PROGRAM Stn055_20_StorageBreakStopsGrn
VAR
	
	//Note that breakstop 1 is controlled by 3 lane swtich so although called a break stop it is not mapped here
	// Remove these outputs temp to avoid common valve bank conflict for control of outputs with station 51
	//	.fbBreakStop[42].oStopLower :=  <0,1,0>TIIB[N13S00 (AL1332)]^N13S02 (EX260)^RxPDO^output byte 0;
	//	.fbBreakStop[43].oStopLower :=  <0,1,1>TIIB[N13S00 (AL1332)]^N13S02 (EX260)^RxPDO^output byte 0'
	
	{attribute 'TcLinkToOSO' := '.fbBreakStop[2].iBufferFull :=  <0,1,1>TIIB[N62S00 (AL1332)]^N62S03 (AL2341)^TxPDO^input byte 2;
		.fbBreakStop[2].iPuckPresent :=  <0,1,1>TIIB[N62S00 (AL1332)]^N62S03 (AL2341)^TxPDO^input byte 0;
		.fbBreakStop[2].oStopLower :=  <0,1,4>TIIB[N62S00 (AL1332)]^N62S02 (EX260)^RxPDO^output byte 0;
		.fbBreakStop[3].iBufferFull :=  <0,1,0>TIIB[N62S00 (AL1332)]^N62S05 (AL2341)^TxPDO^input byte 2;
		.fbBreakStop[3].iPuckPresent :=  <0,1,0>TIIB[N62S00 (AL1332)]^N62S05 (AL2341)^TxPDO^input byte 0;
		.fbBreakStop[3].oStopLower :=  <0,1,5>TIIB[N62S00 (AL1332)]^N62S02 (EX260)^RxPDO^output byte 0;
		.fbBreakStop[4].iBufferFull :=  <0,1,0>TIIB[N66S00 (AL1332)]^N66S01 (AL2341)^TxPDO^input byte 2;
		.fbBreakStop[4].iPuckPresent :=  <0,1,0>TIIB[N66S00 (AL1332)]^N66S01 (AL2341)^TxPDO^input byte 0;
		.fbBreakStop[4].oStopLower :=  <0,1,0>TIIB[N66S00 (AL1332)]^N66S02 (EX260)^RxPDO^output byte 0;
		.fbBreakStop[5].iBufferFull :=  <0,1,1>TIIB[N66S00 (AL1332)]^N66S01 (AL2341)^TxPDO^input byte 2;
		.fbBreakStop[5].iPuckPresent :=  <0,1,1>TIIB[N66S00 (AL1332)]^N66S01 (AL2341)^TxPDO^input byte 0;
		.fbBreakStop[5].oStopLower :=  <0,1,1>TIIB[N66S00 (AL1332)]^N66S02 (EX260)^RxPDO^output byte 0;
		.fbBreakStop[6].iBufferFull :=  <0,1,2>TIIB[N66S00 (AL1332)]^N66S01 (AL2341)^TxPDO^input byte 2;
		.fbBreakStop[6].iPuckPresent :=  <0,1,2>TIIB[N66S00 (AL1332)]^N66S01 (AL2341)^TxPDO^input byte 0;
		.fbBreakStop[6].oStopLower :=  <0,1,2>TIIB[N66S00 (AL1332)]^N66S02 (EX260)^RxPDO^output byte 0;
		.fbBreakStop[7].iBufferFull :=  <0,1,0>TIIB[N66S00 (AL1332)]^N66S03 (AL2341)^TxPDO^input byte 2;
		.fbBreakStop[7].iPuckPresent :=  <0,1,0>TIIB[N66S00 (AL1332)]^N66S03 (AL2341)^TxPDO^input byte 0;
		.fbBreakStop[7].oStopLower :=  <0,1,3>TIIB[N66S00 (AL1332)]^N66S02 (EX260)^RxPDO^output byte 0;
		.fbBreakStop[8].iBufferFull :=  <0,1,1>TIIB[N66S00 (AL1332)]^N66S03 (AL2341)^TxPDO^input byte 2;
		.fbBreakStop[8].iPuckPresent :=  <0,1,1>TIIB[N66S00 (AL1332)]^N66S03 (AL2341)^TxPDO^input byte 0;
		.fbBreakStop[8].oStopLower :=  <0,1,4>TIIB[N66S00 (AL1332)]^N66S02 (EX260)^RxPDO^output byte 0;
		.fbBreakStop[9].iBufferFull :=  <0,1,2>TIIB[N66S00 (AL1332)]^N66S03 (AL2341)^TxPDO^input byte 2;
		.fbBreakStop[9].iPuckPresent :=  <0,1,2>TIIB[N66S00 (AL1332)]^N66S03 (AL2341)^TxPDO^input byte 0;
		.fbBreakStop[9].oStopLower :=  <0,1,5>TIIB[N66S00 (AL1332)]^N66S02 (EX260)^RxPDO^output byte 0;
		.fbBreakStop[10].iBufferFull :=  <0,1,3>TIIB[N66S00 (AL1332)]^N66S03 (AL2341)^TxPDO^input byte 2;
		.fbBreakStop[10].iPuckPresent :=  <0,1,3>TIIB[N66S00 (AL1332)]^N66S03 (AL2341)^TxPDO^input byte 0;
		.fbBreakStop[10].oStopLower :=  <0,1,6>TIIB[N66S00 (AL1332)]^N66S02 (EX260)^RxPDO^output byte 0;
		.fbBreakStop[11].iBufferFull :=  <0,1,0>TIIB[N67S00 (AL1332)]^N67S01 (AL2341)^TxPDO^input byte 2;
		.fbBreakStop[11].iPuckPresent :=  <0,1,0>TIIB[N67S00 (AL1332)]^N67S01 (AL2341)^TxPDO^input byte 0;
		.fbBreakStop[11].oStopLower :=  <0,1,0>TIIB[N67S00 (AL1332)]^N67S02 (EX260)^RxPDO^output byte 0;
		.fbBreakStop[12].iBufferFull :=  <0,1,1>TIIB[N67S00 (AL1332)]^N67S01 (AL2341)^TxPDO^input byte 2;
		.fbBreakStop[12].iPuckPresent :=  <0,1,1>TIIB[N67S00 (AL1332)]^N67S01 (AL2341)^TxPDO^input byte 0;
		.fbBreakStop[12].oStopLower :=  <0,1,1>TIIB[N67S00 (AL1332)]^N67S02 (EX260)^RxPDO^output byte 0;
		.fbBreakStop[13].iBufferFull :=  <0,1,0>TIIB[N67S00 (AL1332)]^N67S01 (AL2341)^TxPDO^input byte 3;
		.fbBreakStop[13].iPuckPresent :=  <0,1,0>TIIB[N67S00 (AL1332)]^N67S01 (AL2341)^TxPDO^input byte 1;
		.fbBreakStop[13].oStopLower :=  <0,1,3>TIIB[N67S00 (AL1332)]^N67S02 (EX260)^RxPDO^output byte 0;
		.fbBreakStop[14].iBufferFull :=  <0,1,1>TIIB[N67S00 (AL1332)]^N67S01 (AL2341)^TxPDO^input byte 3;
		.fbBreakStop[14].iPuckPresent :=  <0,1,1>TIIB[N67S00 (AL1332)]^N67S01 (AL2341)^TxPDO^input byte 1;
		.fbBreakStop[14].oStopLower :=  <0,1,6>TIIB[N67S00 (AL1332)]^N67S02 (EX260)^RxPDO^output byte 0;
		.fbBreakStop[15].iBufferFull :=  <0,1,2>TIIB[N67S00 (AL1332)]^N67S01 (AL2341)^TxPDO^input byte 3;
		.fbBreakStop[15].iPuckPresent :=  <0,1,2>TIIB[N67S00 (AL1332)]^N67S01 (AL2341)^TxPDO^input byte 1;
		.fbBreakStop[15].oStopLower :=  <0,1,7>TIIB[N67S00 (AL1332)]^N67S02 (EX260)^RxPDO^output byte 0;
		.fbBreakStop[16].iBufferFull :=  <0,1,4>TIIB[N67S00 (AL1332)]^N67S03 (AL2341)^TxPDO^input byte 2;
		.fbBreakStop[16].iPuckPresent :=  <0,1,4>TIIB[N67S00 (AL1332)]^N67S03 (AL2341)^TxPDO^input byte 0;
		.fbBreakStop[16].oStopLower :=  <0,1,4>TIIB[N67S00 (AL1332)]^N67S02 (EX260)^RxPDO^output byte 1;
		.fbBreakStop[17].iBufferFull :=  <0,1,1>TIIB[N67S00 (AL1332)]^N67S03 (AL2341)^TxPDO^input byte 3;
		.fbBreakStop[17].iPuckPresent :=  <0,1,1>TIIB[N67S00 (AL1332)]^N67S03 (AL2341)^TxPDO^input byte 1;
		.fbBreakStop[17].oStopLower :=  <0,1,5>TIIB[N67S00 (AL1332)]^N67S02 (EX260)^RxPDO^output byte 1;
		.fbBreakStop[18].iBufferFull :=  <0,1,2>TIIB[N67S00 (AL1332)]^N67S03 (AL2341)^TxPDO^input byte 3;
		.fbBreakStop[18].iPuckPresent :=  <0,1,2>TIIB[N67S00 (AL1332)]^N67S03 (AL2341)^TxPDO^input byte 1;
		.fbBreakStop[18].oStopLower :=  <0,1,0>TIIB[N67S00 (AL1332)]^N67S02 (EX260)^RxPDO^output byte 2;
		.fbBreakStop[19].iBufferFull :=  <0,1,0>TIIB[N67S00 (AL1332)]^N67S05 (AL2341)^TxPDO^input byte 2;
		.fbBreakStop[19].iPuckPresent :=  <0,1,0>TIIB[N67S00 (AL1332)]^N67S05 (AL2341)^TxPDO^input byte 0;
		.fbBreakStop[19].oStopLower :=  <0,1,1>TIIB[N67S00 (AL1332)]^N67S02 (EX260)^RxPDO^output byte 2;
		.fbBreakStop[20].iBufferFull :=  <0,1,1>TIIB[N67S00 (AL1332)]^N67S05 (AL2341)^TxPDO^input byte 2;
		.fbBreakStop[20].iPuckPresent :=  <0,1,1>TIIB[N67S00 (AL1332)]^N67S05 (AL2341)^TxPDO^input byte 0;
		.fbBreakStop[20].oStopLower :=  <0,1,2>TIIB[N67S00 (AL1332)]^N67S02 (EX260)^RxPDO^output byte 2;
		.fbBreakStop[21].iBufferFull :=  <0,1,2>TIIB[N67S00 (AL1332)]^N67S05 (AL2341)^TxPDO^input byte 2;
		.fbBreakStop[21].iPuckPresent :=  <0,1,2>TIIB[N67S00 (AL1332)]^N67S05 (AL2341)^TxPDO^input byte 0;
		.fbBreakStop[21].oStopLower :=  <0,1,3>TIIB[N67S00 (AL1332)]^N67S02 (EX260)^RxPDO^output byte 2;
		.fbBreakStop[22].iBufferFull :=  <0,1,4>TIIB[N67S00 (AL1332)]^N67S05 (AL2341)^TxPDO^input byte 2;
		.fbBreakStop[22].iPuckPresent :=  <0,1,4>TIIB[N67S00 (AL1332)]^N67S05 (AL2341)^TxPDO^input byte 0;
		.fbBreakStop[22].oStopLower :=  <0,1,6>TIIB[N67S00 (AL1332)]^N67S02 (EX260)^RxPDO^output byte 2;
		.fbBreakStop[23].iBufferFull :=  <0,1,0>TIIB[N67S00 (AL1332)]^N67S05 (AL2341)^TxPDO^input byte 3;
		.fbBreakStop[23].iPuckPresent :=  <0,1,0>TIIB[N67S00 (AL1332)]^N67S05 (AL2341)^TxPDO^input byte 1;
		.fbBreakStop[23].oStopLower :=  <0,1,7>TIIB[N67S00 (AL1332)]^N67S02 (EX260)^RxPDO^output byte 2;
		.fbBreakStop[24].iBufferFull :=  <0,1,0>TIIB[N66S00 (AL1332)]^N66S05 (AL2341)^TxPDO^input byte 2;
		.fbBreakStop[24].iPuckPresent :=  <0,1,0>TIIB[N66S00 (AL1332)]^N66S05 (AL2341)^TxPDO^input byte 0;
		.fbBreakStop[24].oStopLower :=  <0,1,0>TIIB[N66S00 (AL1332)]^N66S04 (EX260)^RxPDO^output byte 0;
		.fbBreakStop[25].iBufferFull :=  <0,1,1>TIIB[N66S00 (AL1332)]^N66S05 (AL2341)^TxPDO^input byte 2;
		.fbBreakStop[25].iPuckPresent :=  <0,1,1>TIIB[N66S00 (AL1332)]^N66S05 (AL2341)^TxPDO^input byte 0;
		.fbBreakStop[25].oStopLower :=  <0,1,1>TIIB[N66S00 (AL1332)]^N66S04 (EX260)^RxPDO^output byte 0;
		.fbBreakStop[26].iBufferFull :=  <0,1,2>TIIB[N66S00 (AL1332)]^N66S05 (AL2341)^TxPDO^input byte 2;
		.fbBreakStop[26].iPuckPresent :=  <0,1,2>TIIB[N66S00 (AL1332)]^N66S05 (AL2341)^TxPDO^input byte 0;
		.fbBreakStop[26].oStopLower :=  <0,1,2>TIIB[N66S00 (AL1332)]^N66S04 (EX260)^RxPDO^output byte 0;
		.fbBreakStop[27].iBufferFull :=  <0,1,0>TIIB[N66S00 (AL1332)]^N66S07 (AL2341)^TxPDO^input byte 2;
		.fbBreakStop[27].iPuckPresent :=  <0,1,0>TIIB[N66S00 (AL1332)]^N66S07 (AL2341)^TxPDO^input byte 0;
		.fbBreakStop[27].oStopLower :=  <0,1,3>TIIB[N66S00 (AL1332)]^N66S04 (EX260)^RxPDO^output byte 0;
		.fbBreakStop[28].iBufferFull :=  <0,1,1>TIIB[N66S00 (AL1332)]^N66S07 (AL2341)^TxPDO^input byte 2;
		.fbBreakStop[28].iPuckPresent :=  <0,1,1>TIIB[N66S00 (AL1332)]^N66S07 (AL2341)^TxPDO^input byte 0;
		.fbBreakStop[28].oStopLower :=  <0,1,4>TIIB[N66S00 (AL1332)]^N66S04 (EX260)^RxPDO^output byte 0;
		.fbBreakStop[29].iBufferFull :=  <0,1,0>TIIB[N71S00 (AL1332)]^N71S01 (AL2341)^TxPDO^input byte 2;
		.fbBreakStop[29].iPuckPresent :=  <0,1,0>TIIB[N71S00 (AL1332)]^N71S01 (AL2341)^TxPDO^input byte 0;
		.fbBreakStop[29].oStopLower :=  <0,1,0>TIIB[N71S00 (AL1332)]^N71S02 (EX260)^RxPDO^output byte 0;
		.fbBreakStop[30].iBufferFull :=  <0,1,1>TIIB[N71S00 (AL1332)]^N71S01 (AL2341)^TxPDO^input byte 2;
		.fbBreakStop[30].iPuckPresent :=  <0,1,1>TIIB[N71S00 (AL1332)]^N71S01 (AL2341)^TxPDO^input byte 0;
		.fbBreakStop[30].oStopLower :=  <0,1,1>TIIB[N71S00 (AL1332)]^N71S02 (EX260)^RxPDO^output byte 0;
		.fbBreakStop[31].iBufferFull :=  <0,1,0>TIIB[N71S00 (AL1332)]^N71S03 (AL2341)^TxPDO^input byte 2;
		.fbBreakStop[31].iPuckPresent :=  <0,1,0>TIIB[N71S00 (AL1332)]^N71S03 (AL2341)^TxPDO^input byte 0;
		.fbBreakStop[31].oStopLower :=  <0,1,2>TIIB[N71S00 (AL1332)]^N71S02 (EX260)^RxPDO^output byte 0;
		.fbBreakStop[32].iBufferFull :=  <0,1,1>TIIB[N71S00 (AL1332)]^N71S03 (AL2341)^TxPDO^input byte 2;
		.fbBreakStop[32].iPuckPresent :=  <0,1,1>TIIB[N71S00 (AL1332)]^N71S03 (AL2341)^TxPDO^input byte 0;
		.fbBreakStop[32].oStopLower :=  <0,1,3>TIIB[N71S00 (AL1332)]^N71S02 (EX260)^RxPDO^output byte 0;
		.fbBreakStop[33].iBufferFull :=  <0,1,0>TIIB[N71S00 (AL1332)]^N71S05 (AL2341)^TxPDO^input byte 2;
		.fbBreakStop[33].iPuckPresent :=  <0,1,0>TIIB[N71S00 (AL1332)]^N71S05 (AL2341)^TxPDO^input byte 0;
		.fbBreakStop[33].oStopLower :=  <0,1,4>TIIB[N71S00 (AL1332)]^N71S02 (EX260)^RxPDO^output byte 0;
		.fbBreakStop[34].iBufferFull :=  <0,1,1>TIIB[N71S00 (AL1332)]^N71S05 (AL2341)^TxPDO^input byte 2;
		.fbBreakStop[34].iPuckPresent :=  <0,1,1>TIIB[N71S00 (AL1332)]^N71S05 (AL2341)^TxPDO^input byte 0;
		.fbBreakStop[34].oStopLower :=  <0,1,5>TIIB[N71S00 (AL1332)]^N71S02 (EX260)^RxPDO^output byte 0;
		.fbBreakStop[35].iBufferFull :=  <0,1,0>TIIB[N73S00 (AL1332)]^N73S01 (AL2341)^TxPDO^input byte 2;
		.fbBreakStop[35].iPuckPresent :=  <0,1,0>TIIB[N73S00 (AL1332)]^N73S01 (AL2341)^TxPDO^input byte 0;
		.fbBreakStop[35].oStopLower :=  <0,1,0>TIIB[N73S00 (AL1332)]^N73S02 (EX260)^RxPDO^output byte 0;
		.fbBreakStop[36].iBufferFull :=  <0,1,1>TIIB[N73S00 (AL1332)]^N73S01 (AL2341)^TxPDO^input byte 2;
		.fbBreakStop[36].iPuckPresent :=  <0,1,1>TIIB[N73S00 (AL1332)]^N73S01 (AL2341)^TxPDO^input byte 0;
		.fbBreakStop[36].oStopLower :=  <0,1,1>TIIB[N73S00 (AL1332)]^N73S02 (EX260)^RxPDO^output byte 0;
		.fbBreakStop[37].iBufferFull :=  <0,1,0>TIIB[N73S00 (AL1332)]^N73S03 (AL2341)^TxPDO^input byte 2;
		.fbBreakStop[37].iPuckPresent :=  <0,1,0>TIIB[N73S00 (AL1332)]^N73S03 (AL2341)^TxPDO^input byte 0;
		.fbBreakStop[37].oStopLower :=  <0,1,2>TIIB[N73S00 (AL1332)]^N73S02 (EX260)^RxPDO^output byte 0;
		.fbBreakStop[38].iBufferFull :=  <0,1,1>TIIB[N73S00 (AL1332)]^N73S03 (AL2341)^TxPDO^input byte 2;
		.fbBreakStop[38].iPuckPresent :=  <0,1,1>TIIB[N73S00 (AL1332)]^N73S03 (AL2341)^TxPDO^input byte 0;
		.fbBreakStop[38].oStopLower :=  <0,1,3>TIIB[N73S00 (AL1332)]^N73S02 (EX260)^RxPDO^output byte 0;
		.fbBreakStop[39].iBufferFull :=  <0,1,2>TIIB[N73S00 (AL1332)]^N73S03 (AL2341)^TxPDO^input byte 2;
		.fbBreakStop[39].iPuckPresent :=  <0,1,2>TIIB[N73S00 (AL1332)]^N73S03 (AL2341)^TxPDO^input byte 0;
		.fbBreakStop[39].oStopLower :=  <0,1,4>TIIB[N73S00 (AL1332)]^N73S02 (EX260)^RxPDO^output byte 0;
		.fbBreakStop[40].iBufferFull :=  <0,1,0>TIIB[N73S00 (AL1332)]^N73S05 (AL2341)^TxPDO^input byte 2;
		.fbBreakStop[40].iPuckPresent :=  <0,1,0>TIIB[N73S00 (AL1332)]^N73S05 (AL2341)^TxPDO^input byte 0;
		.fbBreakStop[40].oStopLower :=  <0,1,5>TIIB[N73S00 (AL1332)]^N73S02 (EX260)^RxPDO^output byte 0;
		.fbBreakStop[41].iBufferFull :=  <0,1,1>TIIB[N73S00 (AL1332)]^N73S05 (AL2341)^TxPDO^input byte 2;
		.fbBreakStop[41].iPuckPresent :=  <0,1,1>TIIB[N73S00 (AL1332)]^N73S05 (AL2341)^TxPDO^input byte 0;
		.fbBreakStop[41].oStopLower :=  <0,1,6>TIIB[N73S00 (AL1332)]^N73S02 (EX260)^RxPDO^output byte 0;
		.fbBreakStop[42].iBufferFull :=  <0,1,0>TIIB[N12S00 (AL1332)]^N12S07 (AL2341)^TxPDO^input byte 2;
		.fbBreakStop[42].iPuckPresent :=  <0,1,0>TIIB[N12S00 (AL1332)]^N12S07 (AL2341)^TxPDO^input byte 0;
		.fbBreakStop[43].iBufferFull :=  <0,1,0>TIIB[N13S00 (AL1332)]^N13S01 (AL2341)^TxPDO^input byte 2;
		.fbBreakStop[43].iPuckPresent :=  <0,1,0>TIIB[N13S00 (AL1332)]^N13S01 (AL2341)^TxPDO^input byte 0'}
	fbBreakStopGroup: FB_BreakStopGroup;
	
	i: DINT;
	
END_VAR

//  This code instantiates a component that is implimented as a common function block
//    Note that I/O is linked directly to I/O variables inside the named instance

//  combine running state of any multiple conveyors in a break stop here.
// motor control status here - Green conv 
 
gStn055_20_StorageBreakStopsGrn.ConvRunning[02] := gConsumed_SafetyInterfaceConv.MtrRunning.Enc061Mtr01;
gStn055_20_StorageBreakStopsGrn.ConvRunning[03] := gConsumed_SafetyInterfaceConv.MtrRunning.Enc061Mtr01;
gStn055_20_StorageBreakStopsGrn.ConvRunning[04] := gConsumed_SafetyInterfaceConv.MtrRunning.Enc061Mtr01;
gStn055_20_StorageBreakStopsGrn.ConvRunning[05] := gConsumed_SafetyInterfaceConv.MtrRunning.Enc061Mtr01;
gStn055_20_StorageBreakStopsGrn.ConvRunning[06] := gConsumed_SafetyInterfaceConv.MtrRunning.Enc061Mtr01;
gStn055_20_StorageBreakStopsGrn.ConvRunning[07] := gConsumed_SafetyInterfaceConv.MtrRunning.Enc061Mtr01;
gStn055_20_StorageBreakStopsGrn.ConvRunning[08] := gConsumed_SafetyInterfaceConv.MtrRunning.Enc061Mtr01 AND gConsumed_SafetyInterfaceConv.MtrRunning.Enc061Mtr02;
gStn055_20_StorageBreakStopsGrn.ConvRunning[09] := gConsumed_SafetyInterfaceConv.MtrRunning.Enc061Mtr02;
gStn055_20_StorageBreakStopsGrn.ConvRunning[10] := gConsumed_SafetyInterfaceConv.MtrRunning.Enc061Mtr02;
gStn055_20_StorageBreakStopsGrn.ConvRunning[11] := gConsumed_SafetyInterfaceConv.MtrRunning.Enc061Mtr02;
gStn055_20_StorageBreakStopsGrn.ConvRunning[12] := gConsumed_SafetyInterfaceConv.MtrRunning.Enc061Mtr02;
gStn055_20_StorageBreakStopsGrn.ConvRunning[13] := gConsumed_SafetyInterfaceConv.MtrRunning.Enc061Mtr02;
gStn055_20_StorageBreakStopsGrn.ConvRunning[14] := gConsumed_SafetyInterfaceConv.MtrRunning.Enc061Mtr02;
gStn055_20_StorageBreakStopsGrn.ConvRunning[15] := gConsumed_SafetyInterfaceConv.MtrRunning.Enc061Mtr02 AND gConsumed_SafetyInterfaceConv.MtrRunning.Enc061Mtr04;
gStn055_20_StorageBreakStopsGrn.ConvRunning[16] := gConsumed_SafetyInterfaceConv.MtrRunning.Enc061Mtr04;
gStn055_20_StorageBreakStopsGrn.ConvRunning[17] := gConsumed_SafetyInterfaceConv.MtrRunning.Enc061Mtr04;
gStn055_20_StorageBreakStopsGrn.ConvRunning[18] := gConsumed_SafetyInterfaceConv.MtrRunning.Enc061Mtr04;
gStn055_20_StorageBreakStopsGrn.ConvRunning[19] := gConsumed_SafetyInterfaceConv.MtrRunning.Enc061Mtr04;
gStn055_20_StorageBreakStopsGrn.ConvRunning[20] := gConsumed_SafetyInterfaceConv.MtrRunning.Enc061Mtr04;
gStn055_20_StorageBreakStopsGrn.ConvRunning[21] := gConsumed_SafetyInterfaceConv.MtrRunning.Enc061Mtr04;
gStn055_20_StorageBreakStopsGrn.ConvRunning[22] := gConsumed_SafetyInterfaceConv.MtrRunning.Enc061Mtr04 AND gConsumed_SafetyInterfaceConv.MtrRunning.Enc062Mtr01;
gStn055_20_StorageBreakStopsGrn.ConvRunning[23] := gConsumed_SafetyInterfaceConv.MtrRunning.Enc062Mtr01;
gStn055_20_StorageBreakStopsGrn.ConvRunning[24] := gConsumed_SafetyInterfaceConv.MtrRunning.Enc062Mtr01;
gStn055_20_StorageBreakStopsGrn.ConvRunning[25] := gConsumed_SafetyInterfaceConv.MtrRunning.Enc062Mtr01;
gStn055_20_StorageBreakStopsGrn.ConvRunning[26] := gConsumed_SafetyInterfaceConv.MtrRunning.Enc062Mtr01;
gStn055_20_StorageBreakStopsGrn.ConvRunning[27] := gConsumed_SafetyInterfaceConv.MtrRunning.Enc062Mtr01;
gStn055_20_StorageBreakStopsGrn.ConvRunning[28] := gConsumed_SafetyInterfaceConv.MtrRunning.Enc062Mtr01;
gStn055_20_StorageBreakStopsGrn.ConvRunning[29] := gConsumed_SafetyInterfaceConv.MtrRunning.Enc062Mtr01 AND gConsumed_SafetyInterfaceConv.MtrRunning.Enc062Mtr02;
gStn055_20_StorageBreakStopsGrn.ConvRunning[30] := gConsumed_SafetyInterfaceConv.MtrRunning.Enc062Mtr02;
gStn055_20_StorageBreakStopsGrn.ConvRunning[31] := gConsumed_SafetyInterfaceConv.MtrRunning.Enc062Mtr02;
gStn055_20_StorageBreakStopsGrn.ConvRunning[32] := gConsumed_SafetyInterfaceConv.MtrRunning.Enc062Mtr02;
gStn055_20_StorageBreakStopsGrn.ConvRunning[33] := gConsumed_SafetyInterfaceConv.MtrRunning.Enc062Mtr02;
gStn055_20_StorageBreakStopsGrn.ConvRunning[34] := gConsumed_SafetyInterfaceConv.MtrRunning.Enc062Mtr02;
gStn055_20_StorageBreakStopsGrn.ConvRunning[35] := gConsumed_SafetyInterfaceConv.MtrRunning.Enc062Mtr02;
gStn055_20_StorageBreakStopsGrn.ConvRunning[36] := gConsumed_SafetyInterfaceConv.MtrRunning.Enc062Mtr02 AND gConsumed_SafetyInterfaceConv.MtrRunning.Enc051Mtr01;
gStn055_20_StorageBreakStopsGrn.ConvRunning[37] := gConsumed_SafetyInterfaceConv.MtrRunning.Enc051Mtr01;
gStn055_20_StorageBreakStopsGrn.ConvRunning[38] := gConsumed_SafetyInterfaceConv.MtrRunning.Enc051Mtr01;
gStn055_20_StorageBreakStopsGrn.ConvRunning[39] := gConsumed_SafetyInterfaceConv.MtrRunning.Enc051Mtr01;
gStn055_20_StorageBreakStopsGrn.ConvRunning[40] := gConsumed_SafetyInterfaceConv.MtrRunning.Enc051Mtr01;
gStn055_20_StorageBreakStopsGrn.ConvRunning[41] := gConsumed_SafetyInterfaceConv.MtrRunning.Enc051Mtr01;
gStn055_20_StorageBreakStopsGrn.ConvRunning[42] := gConsumed_SafetyInterfaceConv.MtrRunning.Enc051Mtr01;
gStn055_20_StorageBreakStopsGrn.ConvRunning[43] := gConsumed_SafetyInterfaceConv.MtrRunning.Enc051Mtr01 AND gConsumed_SafetyInterfaceConv.Stn051PLCData[0].10;


fbBreakStopGroup(
	pStn := ADR(gStn055),
	pCmp := ADR(gStn055_20_StorageBreakStopsGrn),
	pStateTraceBuffer := ADR(gStn055_StateTraceBuffer),
	pStateTraceFifo := ADR(gStn055_StateTraceFifo),
	pStats := ADR(gStn055_02_Stats),
);

//Producing lower stop request to station 051 for shared valve bank
gProduced_Stn055ToSafetyInterface.Stn055PLCData[0].0 := gStn055_20_StorageBreakStopsGrn.LowerStopReq[42];
gProduced_Stn055ToSafetyInterface.Stn055PLCData[0].1 := gStn055_20_StorageBreakStopsGrn.LowerStopReq[43];

END_PROGRAM

(* stored: Version 1.1.0.1, ProductVersion 3.1.4024.6
   POU Stn055_20_StorageBreakStopsGrn: Id {58d158b1-18c2-48a1-adad-717d800aeef1}, SpecialFunc None *)
